// TwinCAT 3 PLC project Main
// ProgramVersion: 3.1.4023.0
// libraries:
//   Tc2_DALI, * (Beckhoff Automation GmbH)
//   Tc2_Standard, * (Beckhoff Automation GmbH)
//   Tc2_System, * (Beckhoff Automation GmbH)
//   Tc2_Utilities, * (Beckhoff Automation GmbH)
//   Tc3_IotBase, * (Beckhoff Automation GmbH)
//   Tc3_JsonXml, * (Beckhoff Automation GmbH)
//   Tc3_Module, * (Beckhoff Automation GmbH)
//   BASIC,3.3.3.0,OSCAT
//   BUILDING,1.0.0.0,OSCAT
// project tree:
//   DUTs/Enums/ E_ClickType.TcDUT
//   DUTs/Structs/ ST_ClickTypeCommand.TcDUT, ST_MqttCoverPositionConfiguration.TcDUT, ST_MqttDeviceInformation.TcDUT, ST_MqttDeviceTriggerConfiguration.TcDUT, ST_MqttLightConfiguration.TcDUT
//   GVLs/ GVL_CONST.TcGVL, GVL_MQTT_CONST.TcGVL
//   / PlcTask.TcTTO
//   POUs/Commands/ FB_LightOnCommand.TcPOU, FB_LightOffCommand.TcPOU, FB_LightToggleCommand.TcPOU, FB_MqttDeviceTriggerCommand.TcPOU, FB_MultiCommand_02.TcPOU
//   POUs/FunctionBlocks/ FB_BlindControlS.TcPOU, FB_Light.TcPOU, FB_MqttBlindInputAdapter.TcPOU, FB_MqttLightDecorator.TcPOU, FB_SwitchableDecoratorBase.TcPOU
//   POUs/FunctionBlocks/Homeassistant/Mqtt/ FB_MqttController.TcPOU, FB_MqttCoverPositionDiscovery.TcPOU, FB_MqttDeviceDiscoveryBase.TcPOU, FB_MqttDeviceTriggerDiscovery.TcPOU, FB_MqttLightDiscovery.TcPOU
//   POUs/Functions/ F_StrCmp.TcPOU
//   POUs/Interfaces/ I_Command.TcIO, I_CyclicExecution.TcIO, I_Dimmable.TcIO, I_ClickInvoker.TcIO, I_MqttDeviceDiscovery.TcIO, I_MqttDeviceDiscoveryProvider.TcIO, I_MqttMessageReceiver.TcIO, I_Switchable.TcIO
//   POUs/Invoker/ FB_SwitchClick.TcPOU, FB_ClickPanel2.TcPOU
//   POUs/Programs/ MAIN.TcPOU
// real-time tasks:
//   TASK PlcTask: cycle T#10ms, priority 20, ADS port 350
// I/O:
//   DEVICE Gerät 1 (EtherCAT), AmsNetId 5.68.1.222.2.1
//     Klemme 1 (EK1200) [EK1200-5000 EtherCAT Netzteil (2A E-Bus)]
//       Klemme 2 (EL1252) [EL1252 2K. Fast Dig. Eingang 24V, 1µs, DC Latch]
//       Klemme 3 (EL1252) [EL1252 2K. Fast Dig. Eingang 24V, 1µs, DC Latch]
//       Klemme 4 (EL1252) [EL1252 2K. Fast Dig. Eingang 24V, 1µs, DC Latch]
//       Klemme 5 (EL1252) [EL1252 2K. Fast Dig. Eingang 24V, 1µs, DC Latch]
//       Klemme 6 (EL1252) [EL1252 2K. Fast Dig. Eingang 24V, 1µs, DC Latch]
//       Klemme 7 (EL2252) [EL2252 2K. Dig. Ausgang 24V, 0.5A, DC Time Stamp]
//       Klemme 8 (EL2252) [EL2252 2K. Dig. Ausgang 24V, 0.5A, DC Time Stamp]
//       Klemme 9 (EL2652) [EL2652 2K. Relais Ausgang, Wechsler (230V AC / 30V DC)]
//       Klemme 10 (EL2652) [EL2652 2K. Relais Ausgang, Wechsler (230V AC / 30V DC)]
//       Klemme 11 (EL3112) [EL3112 2K. Ana. Eingang 0-20mA, Diff.]
//       Klemme 12 (EL4112) [EL4112 2K. Ana. Ausgang 0-20mA, 16bit]
//       Klemme 13 (EL9011) [EL9011 Endklemme]
//   DEVICE Gerät 3 (NOV-DP-RAM)
// variable links:
//   Main/Main Instance <-> Device 1 (EtherCAT)/Term 1 (EK1200)/Term 10 (EL2652)
//     PlcTask Outputs/MAIN.bRolloMdn <-> Channel 2/Output
//     PlcTask Outputs/MAIN.bRolloMup <-> Channel 1/Output
//   Main/Main Instance <-> Device 1 (EtherCAT)/Term 1 (EK1200)/Term 2 (EL1252)
//     PlcTask Inputs/MAIN.fbButton1.bSwitch <-> Channel 1/Input
//     PlcTask Inputs/MAIN.fbButton2.bSwitch <-> Channel 2/Input
//   Main/Main Instance <-> Device 1 (EtherCAT)/Term 1 (EK1200)/Term 3 (EL1252)
//     PlcTask Inputs/MAIN.bRolloSdn <-> Channel 2/Input
//     PlcTask Inputs/MAIN.bRolloSup <-> Channel 1/Input
//   Main/Main Instance <-> Device 1 (EtherCAT)/Term 1 (EK1200)/Term 4 (EL1252)
//     PlcTask Inputs/MAIN.bRolloIn <-> Channel 1/Input
//   Main/Main Instance <-> Device 1 (EtherCAT)/Term 1 (EK1200)/Term 9 (EL2652)
//     PlcTask Outputs/MAIN.fbLight.bActive <-> Channel 1/Output

CONFIGURATION Main
    RESOURCE PLC ON TwinCAT3
        TASK PlcTask(INTERVAL := T#10ms, PRIORITY := 20);
        PROGRAM MAIN WITH PlcTask : MAIN;
    END_RESOURCE
END_CONFIGURATION

// ---- DUTs/Enums/E_ClickType.TcDUT
{attribute 'qualified_only'}
{attribute 'strict'}
TYPE E_ClickType :
(
	single := 0,
	double := 1,
	triple := 2,
	longPress := 3,
	longRelease := 4
);
END_TYPE

// ---- DUTs/Structs/ST_ClickTypeCommand.TcDUT
TYPE ST_ClickTypeCommand :
STRUCT
	eClickType: E_ClickType;
	iCommand: I_Command;
END_STRUCT
END_TYPE

// ---- DUTs/Structs/ST_MqttCoverPositionConfiguration.TcDUT
TYPE ST_MqttCoverPositionConfiguration :
STRUCT
	command_topic : STRING(80);
	position_topic : STRING(80);
	set_position_topic : STRING(80);
	payload_open : STRING(10);
	payload_close : STRING(10);
	payload_stop : STRING(10);
	position_open : BYTE;
	position_closed : BYTE;
	device_class: STRING(10);
	optimistic : BOOL;
	unique_id : STRING(20);
	name : STRING(30);
END_STRUCT
END_TYPE

// ---- DUTs/Structs/ST_MqttDeviceInformation.TcDUT
TYPE ST_MqttDeviceInformation :
STRUCT
	// connections: ARRAY[0..1] OF STRING(20); // not working at the moment
	identifiers: STRING(20);
	manufacturer: STRING(20);
	model: STRING(30);
	name: STRING(30);
	sw_version: STRING(10);
	// via_device: STRING(20); // not needed at the moment
END_STRUCT
END_TYPE

// ---- DUTs/Structs/ST_MqttDeviceTriggerConfiguration.TcDUT
(*
	For more information about the valid values of this struct see:
	https://www.home-assistant.io/integrations/device_trigger.mqtt/#configuration-variables
*)
TYPE ST_MqttDeviceTriggerConfiguration :
STRUCT
	payload : STRING(20);		// The payload which shall be sent if the event triggers.
	qos : INT;					// The max qos level to be used for receiving messages.
	topic : STRING(80);			// The events are sent to this topic.
	event_type : STRING(20);	// e.g. button_short_press, button_double_press, ...
	event_subtype : STRING(20); // which button fired (button_1, button_2, ...)
END_STRUCT
END_TYPE

// ---- DUTs/Structs/ST_MqttLightConfiguration.TcDUT
(*
	For more information about the valid values of this struct see:
	https://www.home-assistant.io/integrations/light.mqtt/#configuration-variables
*)
TYPE ST_MqttLightConfiguration :
STRUCT
	command_topic : STRING(80); // to this topic are the commands for on/off sent
	state_topic : STRING(80);	// the light sends state to this topic
	unique_id : STRING(20);		// needed for distinguishment in dev registry
	name : STRING(30);
END_STRUCT
END_TYPE

// ---- GVLs/GVL_CONST.TcGVL
{attribute 'qualified_only'}
VAR_GLOBAL CONSTANT
	SW_VERSION : STRING(10) := '00.00.01';
END_VAR

// ---- GVLs/GVL_MQTT_CONST.TcGVL
{attribute 'qualified_only'}
VAR_GLOBAL
END_VAR
VAR_GLOBAL CONSTANT
	PL_LIGHT_STATE_OFF: STRING(3) := 'OFF';
	DEV_DISCOVER_NODEID : STRING(3) := 'sps';
	DEV_DISCOVER_MANUFACTURER : STRING(10) := 'beckhoff';
	PL_LIGHT_COMMAND_ON: STRING(2) := 'ON';
	PL_LIGHT_COMMAND_OFF: STRING(3) := 'OFF';
	PL_LIGHT_STATE_ON: STRING(2) := 'ON';
	TOPIC_STATE: STRING(10) := 'state';
	TOPIC_COMMAND: STRING(10) := 'set';
	TOPIC_POSITION: STRING(10) := 'position';
	TOPIC_SET_POSITION: STRING(12) := 'set_position';
	PL_COVER_COMMAND_OPEN: STRING(4) := 'OPEN';
	PL_COVER_COMMAND_CLOSE: STRING(5) := 'CLOSE';
	PL_COVER_COMMAND_STOP : STRING(4) := 'STOP';
	COVER_POSITION_OPEN : BYTE := 255;
	COVER_POSITION_CLOSED : BYTE := 0;
	COVER_DEV_CLASS_ROLLO : STRING(10) := 'shutter';
END_VAR

// ---- POUs/Interfaces/I_Command.TcIO
INTERFACE I_Command

METHOD Execute
VAR_INPUT
END_VAR
END_METHOD

END_INTERFACE

// ---- POUs/Interfaces/I_CyclicExecution.TcIO
INTERFACE I_CyclicExecution

METHOD CyclicExecute : BOOL
VAR_INPUT
END_VAR
END_METHOD

END_INTERFACE

// ---- POUs/Interfaces/I_Dimmable.TcIO
INTERFACE I_Dimmable

METHOD GetLevel : BYTE
VAR_INPUT
END_VAR
END_METHOD

METHOD SetLevel : BOOL
VAR_INPUT
	// Level of dimmable
	Level: BYTE := 0;
END_VAR
END_METHOD

END_INTERFACE

// ---- POUs/Interfaces/I_ClickInvoker.TcIO
INTERFACE I_ClickInvoker EXTENDS I_CyclicExecution

METHOD SetCommand : BOOL
VAR_INPUT
	eClickType: E_ClickType; // The Clicktype for which the command shall be registered
	iCmd: I_Command; // The command to be registered
END_VAR
END_METHOD

END_INTERFACE

// ---- POUs/Interfaces/I_MqttDeviceDiscovery.TcIO
INTERFACE I_MqttDeviceDiscovery

METHOD DeleteDevice : BOOL
VAR_INPUT
END_VAR
END_METHOD

PROPERTY DeviceInformation : ST_MqttDeviceInformation
GET
END_GET
END_PROPERTY

PROPERTY NodeId : STRING(20)
GET
END_GET
END_PROPERTY

PROPERTY ObjectId : STRING(40)
GET
END_GET
END_PROPERTY

METHOD RegisterDevice : BOOL
VAR_INPUT
END_VAR
END_METHOD

END_INTERFACE

// ---- POUs/Interfaces/I_MqttDeviceDiscoveryProvider.TcIO
INTERFACE I_MqttDeviceDiscoveryProvider

METHOD GetMqttDeviceDiscovery : I_MqttDeviceDiscovery
VAR_INPUT
END_VAR
END_METHOD

END_INTERFACE

// ---- POUs/Interfaces/I_MqttMessageReceiver.TcIO
INTERFACE I_MqttMessageReceiver

METHOD OnMqttMessage : BOOL
VAR_INPUT
	rMqttMessage : REFERENCE TO FB_IotMqttMessage;
END_VAR
END_METHOD

END_INTERFACE

// ---- POUs/Interfaces/I_Switchable.TcIO
INTERFACE I_Switchable

PROPERTY Active : BOOL
GET
END_GET
END_PROPERTY

METHOD Off : BOOL
VAR_INPUT
END_VAR
END_METHOD

METHOD On : BOOL
VAR_INPUT
END_VAR
END_METHOD

END_INTERFACE

// ---- POUs/Programs/MAIN.TcPOU
PROGRAM MAIN
VAR
	// Communication:
	//fbMqttClient: FB_IotMqttClient;
	fbMqttController : FB_MqttController(sHostname := '192.168.188.13');
	bMqttClientConnect: BOOL := TRUE;
	//fbDevTrigDis : FB_MqttDeviceTriggerDiscovery(fbMqttClient);
	
	// Invokers:
	// The switches ;)
	fbButton1: FB_SwitchClick;
	fbButton2: FB_SwitchClick;
	
	// Receivers:
	// Light in the kitchen
	fbKitchenLight: FB_MqttLightDecorator(
		rMqttController := fbMqttController,
		sMainTopic := 'haus/kueche/esstisch/licht',
		sIdentifier := 'licht_esstisch',
		sName := 'Fressthekenlampe');
	
	// Commands:
	// switching on
	fbKitchenLightOnCommand: FB_LightOnCommand(fbKitchenLight);
	fbKitchenLightOffCommand: FB_LightOffCommand(fbKitchenLight);
	fbKitchenLightToggleCommand: FB_LightToggleCommand(fbKitchenLight);
	fbDevTriggerCommand1: FB_MqttDeviceTriggerCommand(
								rMqttClient := fbMqttController.MqttClient,
								sMainTopic := 'haus/kueche/sw',
								sObjectId := 'sw_kueche_1_single',
								sIdentifier := 'sw_kueche_1',
								sEventType := 'button_short_press',
								sEventSubType := 'button_1',
								sName := 'Schalter 1.1 Kueche Tuere');
	fbDevTriggerCommand2: FB_MqttDeviceTriggerCommand(
								rMqttClient:= fbMqttController.MqttClient,
								sMainTopic := 'haus/kueche/sw',
								sObjectId := 'sw_kueche_1_double',
								sIdentifier := 'sw_kueche_1',
								sEventType := 'button_double_press',
								sEventSubType := 'button_1',
								sName := 'Schalter 1.1 Kueche Tuere');
	arrCmds: ARRAY[0..1] OF I_Command:= [fbDevTriggerCommand1, fbDevTriggerCommand2];
	fbKombiCommand: FB_MultiCommand_02(arrCmds);

	fbMqttBlindAdapter : FB_MqttBlindInputAdapter(
								rMqttController := fbMqttController,
								sMainTopic := 'haus/og/schlafz/cover_l',
								sIdentifier := 'schlafz_l',
								sName := 'Rolladen links');
	fbRolloInput : OSCAT_BUILDING.BLIND_INPUT;
	fbRolloControl : FB_BlindControlS;
	bRolloSup AT %I* : BOOL;
	bRolloSdn AT %I* : BOOL;
	bRolloMup AT %Q* : BOOL;
	bRolloMdn AT %Q* : BOOL;
	bRolloIn AT %I* : BOOL;
	
	// Helpers:
	bInit: BOOL := FALSE;
	bRetVal : BOOL := FALSE;
	bMqttDevicesRegistered : BOOL := FALSE;
END_VAR

IF (NOT bInit) THEN
	fbButton1.SetCommand(E_ClickType.single, fbDevTriggerCommand1);
	fbButton1.SetCommand(E_ClickType.double, fbDevTriggerCommand2);
	
	fbButton2.SetCommand(E_ClickType.single, fbKitchenLightToggleCommand);
	fbButton2.SetCommand(E_ClickType.double, fbKitchenLightOffCommand);
	
	bInit := TRUE;
ELSE
	fbButton1.CyclicExecute();
	fbButton2.CyclicExecute();
	
	fbMqttBlindAdapter(POS := fbRolloControl.POS);
	
	fbRolloInput(POS := fbRolloControl.POS,
		S1 := bRolloSup,
		S2 := bRolloSdn,
		IN := fbMqttBlindAdapter.Q,
		PI := fbMqttBlindAdapter.PO,
		SINGLE_SWITCH := FALSE);
		
	fbRolloControl(UP := fbRolloInput.QU,
		DN := fbRolloInput.QD,
		LOAD := fbMqttBlindAdapter.Q,
		S_IN := fbRolloInput.STATUS,
		PI := fbRolloInput.PO,
		T_UP := T#10S,
		T_DN := T#10S,
		T_EXT := T#2S,
		MU => bRolloMup,
		MD => bRolloMdn);
		
	
END_IF

IF NOT bMqttDevicesRegistered THEN
	bMqttDevicesRegistered := fbDevTriggerCommand1.GetMqttDeviceDiscovery().RegisterDevice();
	IF bMqttDevicesRegistered THEN
		bMqttDevicesRegistered := fbDevTriggerCommand2.GetMqttDeviceDiscovery().RegisterDevice();
	END_IF
	IF bMqttDevicesRegistered THEN
		bMqttDevicesRegistered := fbKitchenLight.GetMqttDeviceDiscovery().RegisterDevice();
	END_IF
	IF bMqttDevicesRegistered THEN
		bMqttDevicesRegistered := fbMqttBlindAdapter.GetMqttDeviceDiscovery().RegisterDevice();
	END_IF
END_IF

fbMqttController.Execute(bMqttClientConnect);

END_PROGRAM

// ---- POUs/FunctionBlocks/Homeassistant/Mqtt/FB_MqttController.TcPOU
FUNCTION_BLOCK FB_MqttController
VAR_INPUT
END_VAR
VAR_OUTPUT
END_VAR
VAR
	fbMqttClient : FB_IotMqttClient;
	fbMqttMsgQueue : FB_IotMqttMessageQueue;
	fbMqttMsg : FB_IotMqttMessage;
	sTopicBuffer : STRING(MAX_TOPIC_LENGTH);
	aMsgTopics : ARRAY[0..MAX_NUM_MSG_RECEIVER - 1] OF STRING(255);
	aMsgReceivers : ARRAY[0..MAX_NUM_MSG_RECEIVER - 1] OF I_MqttMessageReceiver;
	aMsgReceiverValid : ARRAY[0..MAX_NUM_MSG_RECEIVER - 1] OF BOOL;
	bTopicsSubscribed : BOOL;
END_VAR
VAR CONSTANT
	MAX_TOPIC_LENGTH : UINT := 255;
	MAX_NUM_MSG_RECEIVER : UINT := 100;
END_VAR

METHOD Execute : BOOL
VAR_INPUT
	bConnect : BOOL;
END_VAR
VAR
	iMsgReceiver : I_MqttMessageReceiver;
END_VAR
THIS^.fbMqttClient.Execute(bConnect := bConnect);

IF THIS^.fbMqttClient.bConnected AND NOT bTopicsSubscribed THEN
	bTopicsSubscribed := THIS^.SubscribeTopics();
ELSIF NOT THIS^.fbMqttClient.bConnected THEN
	bTopicsSubscribed := FALSE;
END_IF

IF THIS^.fbMqttMsgQueue.nQueuedMessages > 0 THEN
	IF fbMqttMsgQueue.Dequeue(fbMessage := THIS^.fbMqttMsg) THEN
		// search the callback for the topic
		IF fbMqttMsg.GetTopic(pTopic := ADR(THIS^.sTopicBuffer), nTopicSize := MAX_TOPIC_LENGTH) THEN
			IF GetMqttMessageReceiver(sTopic := THIS^.sTopicBuffer, iMsgRcv => iMsgReceiver) THEN
				IF iMsgReceiver <> 0 THEN
					iMsgReceiver.OnMqttMessage(rMqttMessage := fbMqttMsg);
				END_IF
			END_IF
		END_IF
	END_IF
END_IF
END_METHOD

METHOD FB_init : BOOL
VAR_INPUT
	bInitRetains : BOOL; // if TRUE, the retain variables are initialized (warm start / cold start)
	bInCopyCode : BOOL;  // if TRUE, the instance afterwards gets moved into the copy code (online change)
	sHostname : STRING(255);
END_VAR
THIS^.fbMqttClient.sHostName := sHostname;
this^.fbMqttClient.ipMessageQueue := this^.fbMqttMsgQueue;
END_METHOD

METHOD GetMqttMessageReceiver : BOOL
VAR_INPUT
	sTopic : REFERENCE TO STRING(255);
END_VAR
VAR_OUTPUT
	iMsgRcv : I_MqttMessageReceiver;
END_VAR
VAR
	nIndex : UINT;
END_VAR
FOR nIndex := 0 TO MAX_NUM_MSG_RECEIVER - 1 DO
	IF aMsgReceiverValid[nIndex] AND F_StrCmp(pStr1 := ADR(sTopic), pStr2 := ADR(aMsgTopics[nIndex])) THEN
		iMsgRcv := aMsgReceivers[nIndex];
		GetMqttMessageReceiver := TRUE;
		RETURN;
	END_IF
END_FOR

GetMqttMessageReceiver := FALSE;
END_METHOD

PROPERTY MqttClient : REFERENCE TO FB_IotMqttClient
GET
MqttClient REF= this^.fbMqttClient;
END_GET
END_PROPERTY

METHOD RegisterMqttMessageReceive : BOOL
VAR_INPUT
	iMqttMessageReceiver : I_MqttMessageReceiver;
	sTopic : STRING(255);
END_VAR
VAR
	nIndex : UINT;
END_VAR
IF iMqttMessageReceiver <> 0 THEN
	FOR nIndex := 0 TO MAX_NUM_MSG_RECEIVER - 1 DO
		IF NOT aMsgReceiverValid[nIndex] THEN
			aMsgReceivers[nIndex] := iMqttMessageReceiver;
			aMsgTopics[nIndex] := sTopic;
			aMsgReceiverValid[nIndex] := TRUE;
			RegisterMqttMessageReceive := TRUE;
			RETURN;
		END_IF
	END_FOR
END_IF

RegisterMqttMessageReceive := FALSE;
END_METHOD

METHOD SubscribeTopics : BOOL
VAR_INPUT
END_VAR
VAR
	nIndex : UINT;
	bSubscribed : BOOL := FALSE;
END_VAR
FOR nIndex := 0 TO MAX_NUM_MSG_RECEIVER DO
	IF aMsgReceiverValid[nIndex] AND fbMqttClient.bConnected THEN
		bSubscribed := fbMqttClient.Subscribe(sTopic := aMsgTopics[nIndex], eQoS := TcIotMqttQos.AtMostOnceDelivery);
		IF NOT bSubscribed THEN
			SubscribeTopics := FALSE;
			RETURN;
		END_IF
	END_IF
END_FOR

SubscribeTopics := TRUE;
END_METHOD

END_FUNCTION_BLOCK

// ---- POUs/Functions/F_StrCmp.TcPOU
FUNCTION F_StrCmp : BOOL
VAR_INPUT
	pStr1 : POINTER TO BYTE;
	pStr2 : POINTER TO BYTE;
END_VAR
VAR
END_VAR

IF pStr1 = 0 OR pStr2 = 0 THEN
	F_StrCmp := FALSE;
	RETURN;
END_IF

WHILE TRUE DO
	IF pStr1^ <> pStr2^ THEN
		F_StrCmp := FALSE;
		RETURN;
	ELSIF (pStr1^ = 0) AND (pStr2^ = 0) THEN
		F_StrCmp := TRUE;
		RETURN;
	ELSE
		pStr1 := pStr1 + 1;
		pStr2 := pStr2 + 1;
	END_IF 
END_WHILE

END_FUNCTION

// ---- POUs/Invoker/FB_SwitchClick.TcPOU
FUNCTION_BLOCK FB_SwitchClick IMPLEMENTS I_ClickInvoker
VAR_INPUT
	bSwitch AT %I*: BOOL; // The switch which is pressed by the user 
END_VAR
VAR_OUTPUT
END_VAR
VAR
	singleClickCommand: I_Command; // The command to be executed if single click
	doubleClickCommand: I_Command; // The command to be executed if single click
	longPressedCommand: I_Command; // The command to be executed if long Press starts
	longReleasedCommand: I_Command; // The command to be executed if long Press ends
	fbLongReleasedEdge: F_TRIG;
	fbClick: OSCAT_BUILDING.CLICK_MODE;
END_VAR

METHOD CyclicExecute : BOOL
fbClick(in := bSwitch);

IF fbClick.SINGLE THEN
	THIS^.SingleClick();
ELSIF fbClick.DOUBLE THEN
	THIS^.DoubleClick();
ELSIF fbClick.TP_LONG THEN
	THIS^.LongPress();
ELSE
	fbLongReleasedEdge(clk := fbClick.LONG);
	IF fbLongReleasedEdge.Q THEN
		THIS^.LongRelease();
	END_IF
END_IF
END_METHOD

METHOD PROTECTED DoubleClick : BOOL
VAR_INPUT
END_VAR
IF (doubleClickCommand <> 0) THEN
	doubleClickCommand.Execute();
END_IF
END_METHOD

METHOD FB_init : BOOL
VAR_INPUT
	bInitRetains : BOOL; // if TRUE, the retain variables are initialized (warm start / cold start)
	bInCopyCode : BOOL;  // if TRUE, the instance afterwards gets moved into the copy code (online change)
END_VAR
THIS^.singleClickCommand := 0;
THIS^.doubleClickCommand := 0;
THIS^.longPressedCommand := 0;
THIS^.longReleasedCommand := 0;
END_METHOD

METHOD PROTECTED LongPress : BOOL
VAR_INPUT
END_VAR
IF (longPressedCommand <> 0) THEN
	longPressedCommand.Execute();
END_IF
END_METHOD

METHOD PROTECTED LongRelease : BOOL
VAR_INPUT
END_VAR
IF (longReleasedCommand <> 0) THEN
	longReleasedCommand.Execute();
END_IF
END_METHOD

METHOD SetCommand : BOOL
VAR_INPUT
	eClickType: E_ClickType; // The Clicktype for which the command shall be registered
	iCmd: I_Command; // The command to be registered
END_VAR
IF ((eClickType = E_ClickType.single) AND (iCmd <> 0)) THEN
	THIS^.singleClickCommand := iCmd;
	SetCommand := TRUE;
ELSIF ((eClickType = E_ClickType.double) AND (iCmd <> 0)) THEN
	THIS^.doubleClickCommand := iCmd;
	SetCommand := TRUE;
ELSIF ((eClickType = E_ClickType.longPress) AND (iCmd <> 0)) THEN
	THIS^.longPressedCommand := iCmd;
	SetCommand := TRUE;
ELSIF ((eClickType = E_ClickType.longRelease) AND (iCmd <> 0)) THEN
	THIS^.longReleasedCommand := iCmd;
	SetCommand := TRUE;
ELSE
	SetCommand := FALSE;
END_IF
END_METHOD

METHOD PROTECTED SingleClick : BOOL
VAR_INPUT
END_VAR
IF (singleClickCommand <> 0) THEN
	singleClickCommand.Execute();
END_IF
END_METHOD

END_FUNCTION_BLOCK

// ---- POUs/FunctionBlocks/FB_MqttLightDecorator.TcPOU
FUNCTION_BLOCK FB_MqttLightDecorator EXTENDS FB_Light IMPLEMENTS I_MqttMessageReceiver, I_MqttDeviceDiscoveryProvider
VAR_INPUT
END_VAR
VAR_OUTPUT
END_VAR
VAR
	rMqttController: REFERENCE TO FB_MqttController;
	fbDeviceDiscovery : FB_MqttLightDiscovery;
	sStateTopic: STRING(255); // The topic to publish the state to
	sCommandTopic : STRING(255);
	sCmdOnPayload: STRING(10); // The text which is published if On() is called
	sCmdOffPayload: STRING(10); // The test which is published if Off() is called
	sStateOnPayload: STRING(10); // The text which is published if On() is called
	sStateOffPayload: STRING(10); // The test which is published if Off() is called
END_VAR

METHOD FB_init : BOOL
VAR_INPUT
	bInitRetains : BOOL; // if TRUE, the retain variables are initialized (warm start / cold start)
	bInCopyCode : BOOL;  // if TRUE, the instance afterwards gets moved into the copy code (online change)
	rMqttController : REFERENCE TO FB_MqttController;
	sMainTopic : STRING(255); // The topic to publish
	sIdentifier : STRING(20);
	sName : STRING(30);
END_VAR
VAR
	stDevInfo : ST_MqttDeviceInformation;
	stDevConfig : ST_MqttLightConfiguration;
END_VAR
THIS^.rMqttController REF= rMqttController;

THIS^.sStateTopic := CONCAT(STR1 := sMainTopic, STR2 := '/');
THIS^.sStateTopic := CONCAT(STR1 := THIS^.sStateTopic, STR2 := GVL_MQTT_CONST.TOPIC_STATE);
THIS^.sCommandTopic := CONCAT(STR1 := sMainTopic, STR2 := '/');
THIS^.sCommandTopic := CONCAT(STR1 := THIS^.sCommandTopic, STR2 := GVL_MQTT_CONST.TOPIC_COMMAND);

THIS^.fbDeviceDiscovery.SetMqttClient(rMqttClient := THIS^.rMqttController.MqttClient);
THIS^.fbDeviceDiscovery.NodeId := GVL_MQTT_CONST.DEV_DISCOVER_NODEID;
THIS^.fbDeviceDiscovery.ObjectId := sIdentifier;

stDevConfig.command_topic := THIS^.sCommandTopic;
stDevConfig.state_topic := THIS^.sStateTopic;
stDevConfig.unique_id := sIdentifier;
stDevConfig.name := sName;
THIS^.fbDeviceDiscovery.Configuration := stDevConfig;

stDevInfo.identifiers := sIdentifier;
stDevInfo.manufacturer := GVL_MQTT_CONST.DEV_DISCOVER_MANUFACTURER;
stDevInfo.model := 'FB_MqttLight';
stDevInfo.sw_version := GVL_CONST.SW_VERSION;
stDevInfo.name := sName;
THIS^.fbDeviceDiscovery.DeviceInformation := stDevInfo;

THIS^.rMqttController.RegisterMqttMessageReceive(iMqttMessageReceiver := THIS^, sTopic := sCommandTopic);
THIS^.sCmdOnPayload := GVL_MQTT_CONST.PL_LIGHT_COMMAND_ON;
THIS^.sCmdOffPayload := GVL_MQTT_CONST.PL_LIGHT_COMMAND_OFF;
THIS^.sStateOnPayload := GVL_MQTT_CONST.PL_LIGHT_STATE_ON;
THIS^.sStateOffPayload := GVL_MQTT_CONST.PL_LIGHT_STATE_OFF;
END_METHOD

METHOD GetMqttDeviceDiscovery : I_MqttDeviceDiscovery
VAR_INPUT
END_VAR
GetMqttDeviceDiscovery := this^.fbDeviceDiscovery;
END_METHOD

METHOD Off : BOOL
SUPER^.Off();
THIS^.SendStatus();
END_METHOD

METHOD On : BOOL
SUPER^.On();
THIS^.SendStatus();
END_METHOD

METHOD OnMqttMessage : BOOL
VAR_INPUT
	rMqttMessage : REFERENCE TO FB_IotMqttMessage;
END_VAR
VAR
	sPayload : STRING(10);
	bSuccess : BOOL := FALSE;
END_VAR
IF (__ISVALIDREF(rMqttMessage)) THEN
	IF rMqttMessage.GetPayload(pPayload := ADR(sPayload),
			nPayloadSize := 10,
			bSetNullTermination := TRUE) THEN
		IF F_StrCmp(pStr1 := ADR(sPayload), pStr2 := ADR(THIS^.sCmdOnPayload)) THEN
			THIS^.On();
			bSuccess := TRUE;
		ELSIF F_StrCmp(pStr1 := ADR(sPayload), pStr2 := ADR(THIS^.sCmdOffPayload)) THEN
			THIS^.Off();
			bSuccess := TRUE;
		END_IF
	END_IF
END_IF

OnMqttMessage := bSuccess;
END_METHOD

METHOD PRIVATE SendStatus : BOOL
VAR_INPUT
END_VAR
VAR
	sStatus : STRING(10);
END_VAR
IF (__ISVALIDREF(rMqttController) AND __ISVALIDREF(rMqttController.MqttClient)) THEN
	IF (rMqttController.MqttClient.bConnected) THEN
		IF Active THEN
			sStatus := sStateOnPayload;
		ELSE
			sStatus := sStateOffPayload;
		END_IF
		rMqttController.MqttClient.Publish(sTopic:= sStateTopic, 
			pPayload:= ADR(sStatus), nPayloadSize:= LEN2(ADR(sStatus)),
			eQoS:= TcIotMqttQos.AtLeastOnceDelivery, bRetain:= TRUE,
			bQueue:= FALSE);
	END_IF
END_IF
END_METHOD

END_FUNCTION_BLOCK

// ---- POUs/FunctionBlocks/FB_Light.TcPOU
FUNCTION_BLOCK FB_Light IMPLEMENTS I_Switchable
VAR_OUTPUT
	// output of the FB. This is the state of the light.
	bActive AT %Q*: BOOL;
END_VAR

PROPERTY PUBLIC Active : BOOL
GET
Active := bActive;
END_GET
END_PROPERTY

METHOD Off : BOOL
bActive := false;
END_METHOD

METHOD On : BOOL
bActive := true;
END_METHOD

END_FUNCTION_BLOCK

// ---- POUs/FunctionBlocks/Homeassistant/Mqtt/FB_MqttLightDiscovery.TcPOU
FUNCTION_BLOCK FB_MqttLightDiscovery EXTENDS FB_MqttDeviceDiscoveryBase
VAR_INPUT
END_VAR
VAR_OUTPUT
END_VAR
VAR
	stConfig : ST_MqttLightConfiguration;
END_VAR

PROPERTY PROTECTED Component : STRING(30)
GET
Component := 'light';
END_GET
END_PROPERTY

METHOD  ConfigToJson : STRING(1000)
VAR_INPUT
END_VAR
VAR
	fbJsonWriter : FB_JsonSaxWriter;
END_VAR
fbJsonWriter.ResetDocument();
fbJsonWriter.StartObject();
fbJsonWriter.AddKeyString(key := 'cmd_t', value := stConfig.command_topic);
fbJsonWriter.AddKeyString(key := 'stat_t', value := stConfig.state_topic);
fbJsonWriter.AddKeyString(key := 'uniq_id', value := stConfig.unique_id);
fbJsonWriter.AddKeyString(key := 'name', value := stConfig.name);
THIS^.DevInfoToJson(rJsonWriter := fbJsonWriter);
fbJsonWriter.EndObject();
fbJsonWriter.CopyDocument(pDoc := ConfigToJson, nDoc := 1000);
END_METHOD

PROPERTY Configuration : ST_MqttLightConfiguration
GET
Configuration := THIS^.stConfig;
END_GET
SET
this^.stConfig := Configuration;
END_SET
END_PROPERTY

END_FUNCTION_BLOCK

// ---- POUs/FunctionBlocks/Homeassistant/Mqtt/FB_MqttDeviceDiscoveryBase.TcPOU
FUNCTION_BLOCK ABSTRACT FB_MqttDeviceDiscoveryBase IMPLEMENTS I_MqttDeviceDiscovery
VAR_INPUT
END_VAR
VAR_OUTPUT
END_VAR
VAR
	rMqttClient : REFERENCE TO FB_IotMqttClient;
	stDeviceInformation : ST_MqttDeviceInformation;
	sNodeId : STRING(20);
	sObjectId : STRING(40);
END_VAR

PROPERTY PROTECTED ABSTRACT Component : STRING(30)
GET
END_GET
END_PROPERTY

METHOD ABSTRACT ConfigToJson : STRING(1000)
VAR_INPUT
END_VAR
END_METHOD

METHOD DeleteDevice : BOOL
VAR
	sTempTopic : STRING(255) := THIS^.DiscoveryTopic;
END_VAR
IF (__ISVALIDREF(rMqttClient)) THEN
	IF (rMqttClient.bConnected) THEN
		DeleteDevice := rMqttClient.Publish(sTopic := sTempTopic,
			pPayload := 0, nPayloadSize := 0,
			eQos := TcIotMqttQos.AtLeastOnceDelivery, bRetain := TRUE,
			bQueue := FALSE);
	END_IF
END_IF
END_METHOD

PROPERTY DeviceInformation : ST_MqttDeviceInformation
GET
DeviceInformation := this^.stDeviceInformation;
END_GET
SET
this^.stDeviceInformation := DeviceInformation;
END_SET
END_PROPERTY

METHOD PROTECTED DevInfoToJson : BOOL
VAR_INPUT
	rJsonWriter : REFERENCE TO FB_JsonSaxWriter; 
END_VAR
rJsonWriter.AddKey(key := 'dev');
rJsonWriter.StartObject();
(* setting connections is not supported at the moment... 
rJsonWriter.AddKey(key := 'cns');
rJsonWriter.StartArray();
rJsonWriter.AddString(value := stDeviceInformation.connections[0]);
rJsonWriter.AddString(value := stDeviceInformation.connections[1]);
rJsonWriter.EndArray();
*)
rJsonWriter.AddKeyString(key := 'ids', value := stDeviceInformation.identifiers);
rJsonWriter.AddKeyString(key := 'mf', value := stDeviceInformation.manufacturer);
rJsonWriter.AddKeyString(key := 'mdl', value := stDeviceInformation.model);
rJsonWriter.AddKeyString(key := 'name', value := stDeviceInformation.name);
rJsonWriter.AddKeyString(key := 'sw', value := stDeviceInformation.sw_version);
// rJsonWriter.AddKeyString(key := 'via_device', value := stDeviceInformation.via_device);
rJsonWriter.EndObject();
END_METHOD

PROPERTY PROTECTED DiscoveryTopic : STRING(255)
GET
VAR
	sTemp : STRING(255);
END_VAR
sTemp := CONCAT('homeassistant/', THIS^.Component);
sTemp := CONCAT(sTemp, '/');
sTemp := CONCAT(sTemp, THIS^.NodeId);
sTemp := CONCAT(sTemp, '/');
sTemp := CONCAT(sTemp, THIS^.ObjectId);
sTemp := CONCAT(sTemp, '/');
DiscoveryTopic := CONCAT(sTemp, 'config');
END_GET
END_PROPERTY

PROPERTY NodeId : STRING(20)
GET
NodeId := THIS^.sNodeId;
END_GET
SET
THIS^.sNodeId := NodeId;
END_SET
END_PROPERTY

PROPERTY ObjectId : STRING(40)
GET
ObjectId := THIS^.sObjectId;
END_GET
SET
THIS^.sObjectId := ObjectId;
END_SET
END_PROPERTY

METHOD RegisterDevice : BOOL
VAR
	sTempTopic : STRING(255) := THIS^.DiscoveryTopic;
	sConfig : STRING(1000) := THIS^.ConfigToJson();
END_VAR
IF (__ISVALIDREF(rMqttClient)) THEN
	IF (rMqttClient.bConnected) THEN
		RegisterDevice := rMqttClient.Publish(sTopic := sTempTopic,
			pPayload := ADR(sConfig), nPayloadSize := LEN2(ADR(sConfig)),
			eQos := TcIotMqttQos.AtLeastOnceDelivery, bRetain := TRUE,
			bQueue := FALSE);
	END_IF
END_IF
END_METHOD

METHOD PUBLIC SetMqttClient : BOOL
VAR_INPUT
	rMqttClient : REFERENCE TO FB_IotMqttClient;
END_VAR
THIS^.rMqttClient REF= rMqttClient;
END_METHOD

END_FUNCTION_BLOCK

// ---- POUs/Commands/FB_LightOnCommand.TcPOU
FUNCTION_BLOCK FB_LightOnCommand IMPLEMENTS I_Command
VAR_INPUT
END_VAR
VAR_OUTPUT
END_VAR
VAR
	// Reference to the Light that should be switched on.
	iLight: I_Switchable;
END_VAR

METHOD Execute
IF (iLight <> 0) THEN
	THIS^.iLight.On();
END_IF
END_METHOD

METHOD FB_init : BOOL
VAR_INPUT
	bInitRetains : BOOL; // if TRUE, the retain variables are initialized (warm start / cold start)
	bInCopyCode : BOOL;  // if TRUE, the instance afterwards gets moved into the copy code (online change)
	iSwitchable : I_Switchable;
END_VAR
IF (iSwitchable <> 0) THEN
	THIS^.iLight := iSwitchable;
END_IF
END_METHOD

END_FUNCTION_BLOCK

// ---- POUs/Commands/FB_LightOffCommand.TcPOU
FUNCTION_BLOCK FB_LightOffCommand IMPLEMENTS I_Command
VAR_INPUT
END_VAR
VAR_OUTPUT
END_VAR
VAR
	// Reference to the Light that should be switched on.
	iLight: I_Switchable;
END_VAR

METHOD Execute
IF (iLight <> 0) THEN
	THIS^.iLight.Off();
END_IF
END_METHOD

METHOD FB_init : BOOL
VAR_INPUT
	bInitRetains : BOOL; // if TRUE, the retain variables are initialized (warm start / cold start)
	bInCopyCode : BOOL;  // if TRUE, the instance afterwards gets moved into the copy code (online change)
	iSwitchable : I_Switchable;
END_VAR
IF (iSwitchable <> 0) THEN
	THIS^.iLight := iSwitchable;
END_IF
END_METHOD

END_FUNCTION_BLOCK

// ---- POUs/Commands/FB_LightToggleCommand.TcPOU
FUNCTION_BLOCK FB_LightToggleCommand IMPLEMENTS I_Command
VAR_INPUT
END_VAR
VAR_OUTPUT
END_VAR
VAR
	// Reference to the Light that should be switched on.
	iLight: I_Switchable;
	bState: BOOL;
END_VAR

METHOD Execute
IF (iLight <> 0) THEN
	IF (iLight.Active) THEN
		THIS^.iLight.Off();
	ELSE
		THIS^.iLight.On();
	END_IF
END_IF
END_METHOD

METHOD FB_init : BOOL
VAR_INPUT
	bInitRetains : BOOL; // if TRUE, the retain variables are initialized (warm start / cold start)
	bInCopyCode : BOOL;  // if TRUE, the instance afterwards gets moved into the copy code (online change)
	iSwitchable : I_Switchable;
END_VAR
IF (iSwitchable <> 0) THEN
	THIS^.iLight := iSwitchable;
END_IF
END_METHOD

END_FUNCTION_BLOCK

// ---- POUs/Commands/FB_MqttDeviceTriggerCommand.TcPOU
FUNCTION_BLOCK FB_MqttDeviceTriggerCommand IMPLEMENTS I_Command, I_MqttDeviceDiscoveryProvider
VAR_INPUT
END_VAR
VAR_OUTPUT
END_VAR
VAR
	rMqttClient: REFERENCE TO FB_IotMqttClient;
	fbDeviceDiscovery: FB_MqttDeviceTriggerDiscovery;
	sTopic: STRING(255); // topic to publish the payload to
	sPayload: STRING(20); // payload to be published
END_VAR

METHOD Execute
IF (__ISVALIDREF(rMqttClient)) THEN
	IF (rMqttClient.bConnected) THEN
		rMqttClient.Publish(sTopic:= THIS^.sTopic, 
			pPayload:= ADR(THIS^.sPayload), nPayloadSize:= LEN2(ADR(THIS^.sPayload)),
			eQoS:= TcIotMqttQos.AtMostOnceDelivery, bRetain:= TRUE,
			bQueue:= FALSE);
	END_IF
END_IF
END_METHOD

METHOD FB_init : BOOL
VAR_INPUT
	bInitRetains : BOOL; // if TRUE, the retain variables are initialized (warm start / cold start)
	bInCopyCode : BOOL;  // if TRUE, the instance afterwards gets moved into the copy code (online change)
	rMqttClient: REFERENCE TO FB_IotMqttClient;
	sMainTopic: STRING(255);
	sObjectId : STRING(40);
	sIdentifier : STRING(20);
	sEventType: STRING(20);
	sEventSubType: STRING(20); // This string will be added to the topic
	//sPayload: STRING(10);
	sName : STRING(30);
END_VAR
VAR
	stDevInfo : ST_MqttDeviceInformation;
	stDevConfig : ST_MqttDeviceTriggerConfiguration;
	sTemp : STRING(255);
END_VAR
THIS^.rMqttClient REF= rMqttClient;
THIS^.fbDeviceDiscovery.SetMqttClient(rMqttClient := THIS^.rMqttClient);
sTemp := concat(STR1 := sMainTopic, STR2 := '/');
sTemp := concat(STR1 := sTemp, STR2 := sIdentifier);
sTemp := concat(STR1 := sTemp, STR2 := '/');
THIS^.sTopic := CONCAT(STR1 := sTemp, STR2 := sEventSubType);
THIS^.sPayload := sEventType;

THIS^.fbDeviceDiscovery.NodeId := GVL_MQTT_CONST.DEV_DISCOVER_NODEID;
THIS^.fbDeviceDiscovery.ObjectId := sObjectId;
stDevConfig.topic := sTopic;
stDevConfig.payload := sPayload;
stDevConfig.qos := 0;
stDevConfig.event_type := sEventType;
stDevConfig.event_subtype := sEventSubType;
THIS^.fbDeviceDiscovery.Configuration := stDevConfig;
stDevInfo.identifiers := sIdentifier;
stDevInfo.manufacturer := GVL_MQTT_CONST.DEV_DISCOVER_MANUFACTURER;
stDevInfo.model := 'FB_MqttDeviceTriggerCommand';
stDevInfo.sw_version := GVL_CONST.SW_VERSION;
stDevInfo.name := sName;
THIS^.fbDeviceDiscovery.DeviceInformation := stDevInfo;
END_METHOD

METHOD GetMqttDeviceDiscovery : I_MqttDeviceDiscovery
GetMqttDeviceDiscovery := THIS^.fbDeviceDiscovery;
END_METHOD

END_FUNCTION_BLOCK

// ---- POUs/FunctionBlocks/Homeassistant/Mqtt/FB_MqttDeviceTriggerDiscovery.TcPOU
FUNCTION_BLOCK FB_MqttDeviceTriggerDiscovery EXTENDS FB_MqttDeviceDiscoveryBase
VAR_INPUT
END_VAR
VAR_OUTPUT
END_VAR
VAR
	stConfig : ST_MqttDeviceTriggerConfiguration;
END_VAR

PROPERTY PROTECTED Component : STRING(30)
GET
Component := 'device_automation';
END_GET
END_PROPERTY

METHOD  ConfigToJson : STRING(1000)
VAR_INPUT
END_VAR
VAR
	fbJsonWriter : FB_JsonSaxWriter;
END_VAR
fbJsonWriter.ResetDocument();
fbJsonWriter.StartObject();
fbJsonWriter.AddKeyString(key := 'atype', value := 'trigger');
fbJsonWriter.AddKeyString(key := 'pl', value := stConfig.payload);
fbJsonWriter.AddKeyNumber(key := 'qos', value := stConfig.qos);
fbJsonWriter.AddKeyString(key := 't', value := stConfig.topic);
fbJsonWriter.AddKeyString(key := 'type', value := stConfig.event_type);
fbJsonWriter.AddKeyString(key := 'stype', value := stConfig.event_subtype);
THIS^.DevInfoToJson(fbJsonWriter); 
fbJsonWriter.EndObject();
fbJsonWriter.CopyDocument(pDoc := ConfigToJson, nDoc := 1000);
END_METHOD

PROPERTY PUBLIC Configuration : ST_MqttDeviceTriggerConfiguration
GET
Configuration := THIS^.stConfig;
END_GET
SET
THIS^.stConfig := Configuration;
END_SET
END_PROPERTY

END_FUNCTION_BLOCK

// ---- POUs/Commands/FB_MultiCommand_02.TcPOU
FUNCTION_BLOCK FB_MultiCommand_02 IMPLEMENTS I_Command
VAR_INPUT
END_VAR
VAR_OUTPUT
END_VAR
VAR
	arrCommands: ARRAY[0..NUM_OF_COMMANDS - 1] OF I_Command; // The commands to be executed
END_VAR
VAR CONSTANT
	NUM_OF_COMMANDS: INT := 2;
END_VAR

METHOD Execute
VAR
	nIndex: INT;
END_VAR
FOR nIndex := 0 TO NUM_OF_COMMANDS - 1 DO
	IF (arrCommands[nIndex] <> 0) THEN
		arrCommands[nIndex].Execute();
	END_IF
END_FOR
END_METHOD

METHOD FB_init : BOOL
VAR_INPUT
	bInitRetains : BOOL; // if TRUE, the retain variables are initialized (warm start / cold start)
	bInCopyCode : BOOL;  // if TRUE, the instance afterwards gets moved into the copy code (online change)
	arrCmd : ARRAY[0..NUM_OF_COMMANDS - 1] OF I_Command;
END_VAR
VAR
	nIndex : INT;
END_VAR
FOR nIndex := 0 TO (NUM_OF_COMMANDS - 1) DO
	arrCommands[nIndex] := arrCmd[nIndex];
END_FOR
END_METHOD

METHOD SetCommand : BOOL
VAR_INPUT
	nPos : INT;
	iCmd : I_Command;
END_VAR
IF (nPos >= 0) AND (nPos < NUM_OF_COMMANDS) AND (iCmd <> 0) THEN
	arrCommands[nPos] := iCmd;
END_IF
END_METHOD

END_FUNCTION_BLOCK

// ---- POUs/FunctionBlocks/FB_MqttBlindInputAdapter.TcPOU
FUNCTION_BLOCK FB_MqttBlindInputAdapter IMPLEMENTS I_CyclicExecution, I_MqttMessageReceiver, I_MqttDeviceDiscoveryProvider
VAR_INPUT
	POS : BYTE;	// Feedback of blind position
END_VAR
VAR_OUTPUT
	Q : BOOL;  // If new values shall be taken into blind_input. Connect this to "BLIND_INPUT.IN"
	PO : BYTE; // The position values which shall be taken into blind_input. Connect this to "BLIND_INPUT.PI"
END_VAR
VAR
	rMqttController : REFERENCE TO FB_MqttController;
	fbDeviceDiscovery : FB_MqttCoverPositionDiscovery;
	stConfig : ST_MqttCoverPositionConfiguration;
	bSetPositionOutput : BOOL; // var for cycle synchronisation
	tSendPositionUpdatesPeriod : TIME := T#250ms;
	tLastPositionUpdate : TIME := T#0S;
	tCurrent : TIME;
	nLastPositionUpdateValue : BYTE;
	bStopRequested : BOOL;
END_VAR

this^.CyclicExecute();

METHOD Close : BOOL
VAR_INPUT
END_VAR
Close := this^.SetPosition(nPosition := GVL_MQTT_CONST.COVER_POSITION_CLOSED);
END_METHOD

METHOD CyclicExecute : BOOL
THIS^.tCurrent := DWORD_TO_TIME(OSCAT_BASIC.T_PLC_MS());

IF THIS^.bStopRequested THEN
	THIS^.SetPosition(nPosition := THIS^.POS);
	this^.bStopRequested := FALSE;
END_IF

THIS^.Q := THIS^.bSetPositionOutput;
THIS^.bSetPositionOutput := FALSE;

IF THIS^.tCurrent - THIS^.tLastPositionUpdate > THIS^.tSendPositionUpdatesPeriod THEN
	IF THIS^.nLastPositionUpdateValue <> THIS^.POS THEN
		THIS^.SendCurrentPosition();
		THIS^.tLastPositionUpdate := THIS^.tCurrent;
	END_IF
END_IF
END_METHOD

METHOD FB_init : BOOL
VAR_INPUT
	bInitRetains : BOOL; // if TRUE, the retain variables are initialized (warm start / cold start)
	bInCopyCode : BOOL;  // if TRUE, the instance afterwards gets moved into the copy code (online change)
	rMqttController : REFERENCE TO FB_MqttController;
	sMainTopic : STRING(255);
	sIdentifier : STRING(20);
	sName : STRING(30);
END_VAR
VAR
	stDevinfo : ST_MqttDeviceInformation;
	sTemp : STRING(255);
END_VAR
THIS^.rMqttController REF= rMqttController;

THIS^.fbDeviceDiscovery.SetMqttClient(rMqttClient := rMqttController.MqttClient);
THIS^.fbDeviceDiscovery.NodeId := GVL_MQTT_CONST.DEV_DISCOVER_NODEID;
THIS^.fbDeviceDiscovery.ObjectId := sIdentifier;

stDevinfo.identifiers := sIdentifier;
stDevinfo.manufacturer := GVL_MQTT_CONST.DEV_DISCOVER_MANUFACTURER;
stDevinfo.model := 'FB_MqttBlindInputAdapter';
stDevinfo.sw_version := GVL_CONST.SW_VERSION;
stDevinfo.name := sName;
THIS^.fbDeviceDiscovery.DeviceInformation := stDevinfo;

THIS^.stConfig.name := sName;
THIS^.stConfig.device_class := GVL_MQTT_CONST.COVER_DEV_CLASS_ROLLO;
THIS^.stConfig.optimistic := FALSE;
THIS^.stConfig.unique_id := sIdentifier;
sTemp := CONCAT(STR1 := sMainTopic, STR2 := '/');
THIS^.stConfig.command_topic := CONCAT(STR1 := sTemp, STR2 := GVL_MQTT_CONST.TOPIC_COMMAND);
THIS^.stConfig.position_topic := CONCAT(STR1 := sTemp, STR2 := GVL_MQTT_CONST.TOPIC_POSITION);
THIS^.stConfig.set_position_topic := CONCAT(STR1 := sTemp, STR2 := GVL_MQTT_CONST.TOPIC_SET_POSITION);
THIS^.stConfig.payload_close := GVL_MQTT_CONST.PL_COVER_COMMAND_CLOSE;
THIS^.stConfig.payload_open := GVL_MQTT_CONST.PL_COVER_COMMAND_OPEN;
THIS^.stConfig.payload_stop := GVL_MQTT_CONST.PL_COVER_COMMAND_STOP;
THIS^.stConfig.position_closed := GVL_MQTT_CONST.COVER_POSITION_CLOSED;
THIS^.stConfig.position_open := GVL_MQTT_CONST.COVER_POSITION_OPEN;
THIS^.fbDeviceDiscovery.Configuration := THIS^.stConfig;

THIS^.rMqttController.RegisterMqttMessageReceive(
	iMqttMessageReceiver := THIS^,
	sTopic := THIS^.stConfig.command_topic);
THIS^.rMqttController.RegisterMqttMessageReceive(
	iMqttMessageReceiver := THIS^,
	sTopic := THIS^.stConfig.set_position_topic);
END_METHOD

METHOD GetMqttDeviceDiscovery : I_MqttDeviceDiscovery
GetMqttDeviceDiscovery := this^.fbDeviceDiscovery;
END_METHOD

METHOD OnMqttMessage : BOOL
VAR_INPUT
	rMqttMessage	: REFERENCE TO Tc3_IotBase.FB_IotMqttMessage;
END_VAR
VAR
	sPayload : STRING(10);
	nNewPosition : BYTE;
	bSuccess : BOOL := FALSE;
END_VAR
IF (__ISVALIDREF(rMqttMessage)) THEN
	IF rMqttMessage.CompareTopic(sTopic := THIS^.stConfig.command_topic) THEN
		IF rMqttMessage.GetPayload(pPayload := ADR(sPayload),
				nPayloadSize := 10,
				bSetNullTermination := TRUE) THEN
			IF F_StrCmp(pStr1 := ADR(sPayload), pStr2 := ADR(THIS^.stConfig.payload_close)) THEN
				THIS^.Close();
				bSuccess := TRUE;
			ELSIF F_StrCmp(pStr1 := ADR(sPayload), pStr2 := ADR(THIS^.stConfig.payload_open)) THEN
				THIS^.Open();
				bSuccess := TRUE;
			ELSIF F_StrCmp(pStr1 := ADR(sPayload), pStr2 := ADR(THIS^.stConfig.payload_stop)) THEN
				THIS^.Stop();
				bSuccess := TRUE;
			END_IF
		END_IF
	ELSIF rMqttMessage.CompareTopic(sTopic := THIS^.stConfig.set_position_topic) THEN
		IF rMqttMessage.GetPayload(pPayload := ADR(sPayload),
				nPayloadSize := 10,
				bSetNullTermination := TRUE) THEN
			nNewPosition := OSCAT_BASIC.DEC_TO_BYTE(DEC := sPayload);
			bSuccess := THIS^.SetPosition(nPosition := nNewPosition);
		END_IF
	END_IF
END_IF

OnMqttMessage := bSuccess;
END_METHOD

METHOD Open : BOOL
VAR_INPUT
END_VAR
Open := this^.SetPosition(nPosition := GVL_MQTT_CONST.COVER_POSITION_OPEN);
END_METHOD

METHOD PRIVATE SendCurrentPosition : BOOL
VAR_INPUT
END_VAR
VAR
	nPositionValue : BYTE;
	sPosValue : STRING(4);
END_VAR
IF (__ISVALIDREF(rMqttController) AND __ISVALIDREF(rMqttController.MqttClient)) THEN
	IF (rMqttController.MqttClient.bConnected) THEN
		nPositionValue := THIS^.POS;
		sPosValue := BYTE_TO_DECSTR(in := nPositionValue, iPrecision := 1);
		SendCurrentPosition := rMqttController.MqttClient.Publish(sTopic:= THIS^.stConfig.position_topic, 
			pPayload:= ADR(sPosValue), nPayloadSize:= LEN2(ADR(sPosValue)),
			eQoS:= TcIotMqttQos.AtMostOnceDelivery, bRetain:= TRUE,
			bQueue:= FALSE);
		IF SendCurrentPosition THEN
			THIS^.nLastPositionUpdateValue := nPositionValue;
		END_IF
	END_IF
END_IF
END_METHOD

METHOD SetPosition : BOOL
VAR_INPUT
	nPosition : BYTE;
END_VAR
THIS^.PO := nPosition;
THIS^.bSetPositionOutput := TRUE;
SetPosition := TRUE;
END_METHOD

METHOD Stop : BOOL
VAR_INPUT
END_VAR
THIS^.bStopRequested := TRUE;
Stop := TRUE;
END_METHOD

END_FUNCTION_BLOCK

// ---- POUs/FunctionBlocks/Homeassistant/Mqtt/FB_MqttCoverPositionDiscovery.TcPOU
FUNCTION_BLOCK FB_MqttCoverPositionDiscovery EXTENDS FB_MqttDeviceDiscoveryBase
VAR_INPUT
END_VAR
VAR_OUTPUT
END_VAR
VAR
	stConfig : ST_MqttCoverPositionConfiguration;
END_VAR

PROPERTY PROTECTED Component : STRING(30)
GET
Component := 'cover';
END_GET
END_PROPERTY

METHOD  ConfigToJson : STRING(1000)
VAR_INPUT
END_VAR
VAR
	fbJsonWriter : FB_JsonSaxWriter;
END_VAR
fbJsonWriter.ResetDocument();
fbJsonWriter.StartObject();
fbJsonWriter.AddKeyString(key := 'cmd_t', value := THIS^.stConfig.command_topic);
fbJsonWriter.AddKeyString(key := 'pos_t', value := THIS^.stConfig.position_topic);
fbJsonWriter.AddKeyString(key := 'set_pos_t', value := THIS^.stConfig.set_position_topic);
fbJsonWriter.AddKeyString(key := 'pl_open', value := THIS^.stConfig.payload_open);
fbJsonWriter.AddKeyString(key := 'pl_cls', value := THIS^.stConfig.payload_close);
fbJsonWriter.AddKeyString(key := 'pl_stop', value := THIS^.stConfig.payload_stop);
fbJsonWriter.AddKeyNumber(key := 'pos_open', value := THIS^.stConfig.position_open);
fbJsonWriter.AddKeyNumber(key := 'pos_clsd', value := THIS^.stConfig.position_closed);
fbJsonWriter.AddKeyString(key := 'dev_cla', value := THIS^.stConfig.device_class);
fbJsonWriter.AddKeyBool(key := 'opt', value := THIS^.stConfig.optimistic);
fbJsonWriter.AddKeyString(key := 'uniq_id', value := THIS^.stConfig.unique_id);
fbJsonWriter.AddKeyString(key := 'name', value := this^.stConfig.name);
THIS^.DevInfoToJson(rJsonWriter := fbJsonWriter);
fbJsonWriter.EndObject();
fbJsonWriter.CopyDocument(pDoc := ConfigToJson, nDoc := 1000);
END_METHOD

PROPERTY Configuration : ST_MqttCoverPositionConfiguration
GET
Configuration := this^.stConfig;
END_GET
SET
this^.stConfig := Configuration;
END_SET
END_PROPERTY

END_FUNCTION_BLOCK

// ---- POUs/FunctionBlocks/FB_BlindControlS.TcPOU
FUNCTION_BLOCK FB_BlindControlS
VAR_INPUT
	UP, DN : BOOL;
	S_IN : BYTE := 125;
	PI : BYTE;
	T_UP : TIME;
	T_DN : TIME;
	RU : BOOL;
	RD : BOOL;
	LOAD : BOOL;		// Load current value in PI.
END_VAR
VAR_INPUT CONSTANT
	T_LOCKOUT: TIME := T#100ms;
	T_EXT : TIME;
	EXT_TRIG : BYTE := 5;
	R_POS_TOP : BYTE := 255;
	R_POS_BOT : BYTE;
END_VAR
VAR_OUTPUT
	POS : BYTE;
	MU, MD : BOOL;
	STATUS : BYTE;
END_VAR
VAR
	rmp : OSCAT_BASIC._RMP_NEXT;
	tx, last : TIME;
	PI_last: BYTE;
END_VAR


(*
version 1.2	23. jan 2010
programmer 	hugo
tested by		heinz


*)


(* status definition
	121 = manual up				manual up operation UP = true and DN = false
	122 = manual down			manual down operation DN = true and UP = false
	123 = auto positioning		automatic mode DN = UP = TRUE
	124 = revert					revert from top or bottom
	125 = nothing					default input for S_IN
	127 = Lockout time			lockout between directional change
	128 = calibrate				calibrate after power up
	129 = extend					extend runtime at top or bottom for continuous calibration
*)

(* read system time *)
tx := DWORD_TO_TIME(OSCAT_BASIC.T_PLC_MS());

(* check inputs and start state machine *)
IF UP  AND NOT DN THEN
	(*  manual UP *)
	rmp.IN := 255;
	STATUS := 121;
ELSIF DN AND NOT UP THEN
	(* manual DN *)
	rmp.IN := 0;
	STATUS := 122;
ELSIF NOT (UP OR DN) THEN
	(* manual standby mode *)
	rmp.IN := PI;
	STATUS := S_IN;
ELSE
	(* auto mode *)
	IF LOAD THEN
		rmp.IN := PI;
	END_IF
END_IF;

(* simulate pos output *)
rmp(E := UP OR DN, TR := T_UP, TF := T_DN, TL := T_LOCKOUT, OUT := POS);

(* state machine *)
CASE STATUS OF
	0:		(* power up init *)
		last := tx;
		PI_last := PI XOR BYTE#255;
		STATUS := 128;		(* calibrate *)

	121: 	(* manual up *)
		MU := TRUE;
		MD := FALSE;
		IF POS >= (BYTE#255 - EXT_TRIG) THEN
			(* extend cycle if top is reached *)
			POS := 255;
			last := tx;
			STATUS := 129;	(* extend *)
		END_IF;

	122:	(* manual down *)
		MD := TRUE;
		MU := FALSE;
		IF POS <= EXT_TRIG THEN
			(* extend cycle if bottom is reached *)
			POS := 0;
			last := tx;
			STATUS := 129;	(* extend *)
		END_IF;

	123:	(* auto positioning *)
		MD := rmp.DN;
		MU := rmp.UP;
		IF NOT (rmp.DN OR rmp.UP) THEN
			(* automatic position is reached *)
			IF POS <= EXT_TRIG THEN
				(* extend at bottom *)
				MD := TRUE;
				last := tx;
				STATUS := 129;	(* extend *)
			ELSIF POS >= (BYTE#255 - EXT_TRIG)  THEN
				(* extend at top *)
				MU := TRUE;
				last := tx;
				STATUS := 129;	(* extend *)
			ELSE
				STATUS := S_IN;
			END_IF;
		END_IF;

	124:	(* revert from top or bottom *)
		MD := rmp.DN;
		MU := rmp.UP;
		IF NOT(rmp.DN OR rmp.UP) THEN
(*		IF POS = rmp.IN THEN  *)
			PI_last := PI;
			STATUS := S_IN;
		END_IF;

	127:	(* lockout time *)
		IF (tx - last) >= T_LOCKOUT THEN
				STATUS := S_IN;
		END_IF;

	128:	(* calibration *)
		MU := TRUE;
		MD := FALSE;
		rmp.IN := 255;
		IF (tx - last) >= (T_UP +  T_EXT) THEN
			MU := FALSE;
			last := tx;
			STATUS := 127;	(* lockout *)
		END_IF;

	129: (* extend mode *)
		IF (tx - last) >= T_EXT THEN
			MU := FALSE;
			MD := FALSE;
			last := tx;
			STATUS := 127;	(* lockout *)
		END_IF;

ELSE
	MU := FALSE;
	MD := FALSE;
	IF PI <> PI_last THEN
		PI_last := PI;
		rmp.IN := PI;
		STATUS := 123;	(* auto positioning *)
	ELSIF POS = 0 AND RU THEN
		rmp.IN := R_POS_BOT;
		STATUS := 124;	(* revert *)
	ELSIF pos = 255 AND RD THEN
		rmp.IN := R_POS_TOP;
		STATUS := 124;	(* revert *)
	ELSE
		STATUS := S_IN;
	END_IF;
END_CASE;



(* revision history

hm	9. mar. 2009	rev 1.0
	original release

hf	27. jul 2009	rev 1.1
	major code changes and updates

hf	23. Jan 2010	rev 1.2
	fixed a bug during calibration
	added T_UP and T_DN

*)

END_FUNCTION_BLOCK

// ---- POUs/FunctionBlocks/FB_SwitchableDecoratorBase.TcPOU
FUNCTION_BLOCK FB_SwitchableDecoratorBase IMPLEMENTS I_Switchable
VAR_INPUT
END_VAR
VAR_OUTPUT
END_VAR
VAR
	iSwitchable : I_Switchable;
END_VAR

PROPERTY Active : BOOL
GET
END_GET
END_PROPERTY

METHOD FB_init : BOOL
VAR_INPUT
	bInitRetains : BOOL; // if TRUE, the retain variables are initialized (warm start / cold start)
	bInCopyCode : BOOL;  // if TRUE, the instance afterwards gets moved into the copy code (online change)
	iSwitchable : I_Switchable; // The switchable to be decorated.
END_VAR
this^.iSwitchable := iSwitchable;
END_METHOD

METHOD Off : BOOL
END_METHOD

METHOD On : BOOL
END_METHOD

PROPERTY PUBLIC Switchable : BOOL
GET
Switchable := THIS^.iSwitchable;
END_GET
SET
THIS^.iSwitchable := Switchable;
END_SET
END_PROPERTY

END_FUNCTION_BLOCK

// ---- POUs/Invoker/FB_ClickPanel2.TcPOU
FUNCTION_BLOCK FB_ClickPanel2
VAR_INPUT
END_VAR
VAR
	arrIClickInvoker: ARRAY[0..1] OF I_ClickInvoker; // The switches of this panel
	nIndex: INT; // Looping helper
END_VAR

FOR nIndex := 0 TO 1 DO
	arrIClickInvoker[nIndex].CyclicExecute();
END_FOR

METHOD FB_init : BOOL
VAR_INPUT
	bInitRetains : BOOL; // if TRUE, the retain variables are initialized (warm start / cold start)
	bInCopyCode : BOOL;  // if TRUE, the instance afterwards gets moved into the copy code (online change)
	arrIClickInvoker : ARRAY[0..1] OF I_ClickInvoker; // The invokers
END_VAR
FOR nIndex := 0 TO 1 DO
	this^.arrIClickInvoker[nIndex] := arrIClickInvoker[nIndex];
END_FOR
END_METHOD

METHOD SetClickInvoker : BOOL
VAR_INPUT
	nPos : INT; // Position of the Clickinvoker
	iClickInvoker : I_ClickInvoker; // the invoker itself...
END_VAR
IF (nPos >= 0) AND (nPos <= 1) AND (iClickInvoker <> 0) THEN
	THIS^.arrFbSwitchClick[nPos] := iClickInvoker;
	SetClickInvoker := TRUE;
ELSE
	SetClickInvoker := FALSE;
END_IF
END_METHOD

METHOD PUBLIC SetCommand : BOOL
VAR_INPUT
	nPosition: INT;				// The position of the switch button
	eClickType: E_ClickType;	// The Clicktype for which the command shall be set
	iCmd: I_Command;			// The command to be set to position nPosition
END_VAR
IF ((nPosition >= 0) AND (nPosition <= 1) AND (iCmd <> 0)) THEN
	THIS^.arrIClickInvoker[nPosition].SetCommand(eClickType := eClickType, iCmd := iCmd);
END_IF
END_METHOD

END_FUNCTION_BLOCK
